Staubli VAL3: INIT.pgx

public program Init()
begin

end
